// TwinCAT 3 PLC project PLC
// ProgramVersion: 3.1.4024.0
// libraries:
//   SPT Base Types, * (Beckhoff Automation LLC)
//   SPT Event Logger, * (Beckhoff Automation LLC)
//   Tc2_Standard, * (Beckhoff Automation GmbH)
//   Tc2_System, * (Beckhoff Automation GmbH)
//   Tc3_EventLogger, * (Beckhoff Automation GmbH)
//   Tc3_Module, * (Beckhoff Automation GmbH)
//   Tc3_PackML_V2, * (Beckhoff Automation GmbH)
// project tree:
//   / PlcTask.TcTTO (not stored)
//   POUs/ Component.TcPOU, EquipmentModule.TcPOU, EquipmentModuleWithSubModule.TcPOU, Machine.TcPOU, MAIN.TcPOU
// real-time tasks:
//   TASK PlcTask: cycle T#10ms, priority 20, ADS port 350

// ---- POUs/Component.TcPOU
FUNCTION_BLOCK Component EXTENDS FB_ComponentBase
VAR
	ComponentAlarms : ARRAY[1..COMPONENT_ALARM_COUNT] OF FB_TcAlarm;
	testCritical	: BOOL;
	testError		: BOOL;
	testWarning		: BOOL;
	testInfo		: BOOL;
	testVerbose		: BOOL;
	clearAlarms		: BOOL;
	testAnalog		: BOOL;
	AnalogIn		: INT;
END_VAR

VAR CONSTANT
	COMPONENT_ALARM_COUNT : UDINT := 7; //First is InitReferenceEvent
END_VAR

METHOD ChangeEventSeverity
VAR_INPUT
	AlarmID : E_ComponentEvents;
	Severity : TcEventSeverity;
END_VAR
VAR
	localAlarm : TcEventEntry;
END_VAR
localAlarm			 := TC_EVENTS.ComponentEvents.AnalogInAlarm;
localAlarm.eSeverity := Severity;
ComponentAlarms[AlarmID].CreateEx(localAlarm, 0, 0);
END_METHOD

//! @summary Initializes event function blocks using this components's name
METHOD PROTECTED CreateEvents

//! @description This method is called by <c>Initialize()</c> as required
F_CreateAllEventsInClass(Alarms		:= ComponentAlarms,
						 ClassSize	:= SIZEOF(TC_Events.ComponentEvents),
						 pInitEvent := ADR(TC_EVENTS.ComponentEvents.InitReferenceEvent),
						 Prefix		:= Name);

SUPER^.CreateEvents();
END_METHOD

//! @summary This method serves as the entry point for all underlying FB logic
METHOD PUBLIC CyclicLogic

//! @description This method should be called cyclically by descendant function blocks by invoking <c>SUPER^.CyclicLogic()</c>.  Alternatively, the contents of this method could be reimplemented entirely in which case a call to this method would not be necessary.
VAR

END_VAR
IF NOT _InitComplete THEN
	_InitComplete := Initialize();
	RETURN;
END_IF



SUPER^.CyclicLogic();

(*
*
*		Code must be after SUPER^.CyclicLogic();
*
*)

(* Update alarm severity from this component *)
_CurrentAlarmSeverity := F_GetMaxSeverityRaised(Alarms := ComponentAlarms, CurrentSeverity := _CurrentAlarmSeverity);
_Error				  := _CurrentAlarmSeverity >= TcEventSeverity.Error;
END_METHOD

//! @summary Basic component initialization logic
METHOD PROTECTED Initialize : BOOL;

//! @description This method is called by <c>CyclicLogic()</c> as required
Initialize := SUPER^.Initialize();
END_METHOD

//! Provides basic error detection and event handling for this component
METHOD PROTECTED Monitoring

(*! @descriptionThis method is called cyclically by <c>CyclicLogic()</c>*)
VAR

END_VAR
_Busy := FALSE;

//AlarmMonitoring
IF testVerbose AND NOT ComponentAlarms[E_ComponentEvents.VerboseEvent].bRaised THEN
	RaiseAlarm2Args(ComponentAlarms[E_ComponentEvents.VerboseEvent], 'Note 1', 'Note 2');
END_IF

IF testInfo AND NOT ComponentAlarms[E_ComponentEvents.InfoEvent].bRaised THEN
	RaiseAlarm2Args(ComponentAlarms[E_ComponentEvents.InfoEvent], 'Note 1', 'Note 2');
END_IF

IF testWarning AND NOT ComponentAlarms[E_ComponentEvents.WarningEvent].bRaised THEN
	RaiseAlarm2Args(ComponentAlarms[E_ComponentEvents.WarningEvent], 'Note 1', 'Note 2');
END_IF

IF testError AND NOT ComponentAlarms[E_ComponentEvents.ErrorEvent].bRaised THEN
	RaiseAlarm2Args(ComponentAlarms[E_ComponentEvents.ErrorEvent], 'Note 1', 'Note 2');
END_IF

IF testCritical AND NOT ComponentAlarms[E_ComponentEvents.CriticalEvent].bRaised THEN
	RaiseAlarm2Args(ComponentAlarms[E_ComponentEvents.CriticalEvent], 'Note 1', 'Note 2');
END_IF

//Analog Input with Changing Event Severities
IF testAnalog AND NOT ComponentAlarms[E_ComponentEvents.AnalogInAlarm].bRaised THEN
	CASE AnalogIn OF
		0..10:
			ChangeEventSeverity(E_ComponentEvents.AnalogInAlarm, TcEventSeverity.Critical);

		11..100:
			ChangeEventSeverity(E_ComponentEvents.AnalogInAlarm, TcEventSeverity.Error);

		101..999:
			ChangeEventSeverity(E_ComponentEvents.AnalogInAlarm, TcEventSeverity.Info);

		1000..1100:
			ChangeEventSeverity(E_ComponentEvents.AnalogInAlarm, TcEventSeverity.Error);

		1101..1201:
			ChangeEventSeverity(E_ComponentEvents.AnalogInAlarm, TcEventSeverity.Critical);
	END_CASE

	RaiseAlarm2Args(ComponentAlarms[E_ComponentEvents.AnalogInAlarm], 'Analong Input:', TO_STRING(AnalogIn));
ELSIF NOT testAnalog AND_THEN ComponentAlarms[E_ComponentEvents.AnalogInAlarm].bRaised THEN
	ComponentAlarms[E_ComponentEvents.AnalogInAlarm].Clear(0, 0);
END_IF

SUPER^.Monitoring();
END_METHOD

METHOD RaiseAlarm2Args
VAR_IN_OUT
	Alarm : FB_TcAlarm; //Alarm to be raised
END_VAR

VAR_INPUT
	String_1 : STRING; //First String Parameter (The Name of this component will be applied first automatically)
	String_2 : STRING; //Second String Parameter
END_VAR
F_RaiseAlarmWithStringParameters(Alarm	  := Alarm,
								 String_1 := Name,
								 String_2 := String_1,
								 String_3 := String_2);
END_METHOD

//! @summary Clears error flags and error IDs for this component
//Typically called by the EMs SUPER^.Clearing Method
METHOD PUBLIC Reset : BOOL
F_ClearAllEventsInClass(Alarms := ComponentAlarms);
IF SUPER^.Reset() THEN
	_Error	 := FALSE;
	_ErrorID := 0;
	Reset	 := TRUE;
END_IF
END_METHOD

END_FUNCTION_BLOCK

// ---- POUs/EquipmentModule.TcPOU
FUNCTION_BLOCK EquipmentModule EXTENDS FB_PackML_BaseModule
VAR
	//Component
	ComponentOne	: Component := (Name := 'Component One');
	EquipmentAlarms : ARRAY[1..EQUIPMENT_ALARM_COUNT] OF FB_TcAlarm;
	testCritical	: BOOL;
	testError		: BOOL;
	testWarning		: BOOL;
	testInfo		: BOOL;
	testVerbose		: BOOL;
	clearAlarms		: BOOL;

END_VAR

VAR CONSTANT
	EQUIPMENT_ALARM_COUNT : UDINT := 6; //First is InitReferenceEvent
END_VAR

METHOD PROTECTED Clearing
VAR
	i				: UDINT;
	SubModulesReady : BOOL := TRUE;
END_VAR
F_ClearAllEventsInClass(Alarms := EquipmentAlarms);
SUPER^.Clearing();
END_METHOD

//! @summary Initializes event function blocks using this module's name
METHOD PROTECTED CreateEvents

//! @description This method is called by <c>Initialize()</c> as required
F_CreateAllEventsInClass(Alarms		:= EquipmentAlarms,
						 ClassSize	:= SIZEOF(TC_Events.EquipmentModuleEvents),
						 pInitEvent := ADR(TC_EVENTS.EquipmentModuleEvents.InitReferenceEvent),
						 Prefix		:= Name);

SUPER^.CreateEvents();
END_METHOD

//! @summary This method serves as the entry point for all underlying FB logic

//! @description This method should be called cyclically by descendant function blocks by invoking <c>SUPER^.CyclicLogic()</c>.  Alternatively, the contents of this method could be reimplemented entirely in which case a call to this method would not be necessary.
METHOD PUBLIC CyclicLogic
VAR
	i : UDINT;
END_VAR
IF NOT _InitComplete THEN
	_InitComplete := Initialize();
	RETURN;
END_IF

//AlarmHandling();
IF testVerbose AND_THEN NOT EquipmentAlarms[E_EquipmentModuleEvents.VerboseEvent].bRaised THEN
	RaiseAlarm2Args(EquipmentAlarms[E_EquipmentModuleEvents.VerboseEvent], 'Note 1', 'Note 2');
ELSIF NOT testVerbose AND_THEN EquipmentAlarms[E_EquipmentModuleEvents.VerboseEvent].bRaised THEN
	EquipmentAlarms[E_EquipmentModuleEvents.VerboseEvent].Clear(0,0);
END_IF

IF testInfo AND_THEN NOT EquipmentAlarms[E_EquipmentModuleEvents.InfoEvent].bRaised THEN
	RaiseAlarm2Args(EquipmentAlarms[E_EquipmentModuleEvents.InfoEvent], 'Note 1', 'Note 2');
ELSIF NOT testInfo AND_THEN EquipmentAlarms[E_EquipmentModuleEvents.InfoEvent].bRaised THEN
	EquipmentAlarms[E_EquipmentModuleEvents.InfoEvent].Clear(0,0);
END_IF

IF testWarning AND_THEN NOT EquipmentAlarms[E_EquipmentModuleEvents.WarningEvent].bRaised THEN
	RaiseAlarm2Args(EquipmentAlarms[E_EquipmentModuleEvents.WarningEvent], 'Note 1', 'Note 2');
ELSIF NOT testWarning AND_THEN EquipmentAlarms[E_EquipmentModuleEvents.WarningEvent].bRaised THEN
	EquipmentAlarms[E_EquipmentModuleEvents.WarningEvent].Clear(0,0);
END_IF

IF testError AND_THEN NOT EquipmentAlarms[E_EquipmentModuleEvents.ErrorEvent].bRaised THEN
	RaiseAlarm2Args(EquipmentAlarms[E_EquipmentModuleEvents.ErrorEvent], 'Note 1', 'Note 2');
END_IF

IF testCritical AND_THEN NOT EquipmentAlarms[E_EquipmentModuleEvents.CriticalEvent].bRaised THEN
	RaiseAlarm2Args(EquipmentAlarms[E_EquipmentModuleEvents.CriticalEvent], 'Note 1', 'Note 2');
END_IF

SUPER^.CyclicLogic();

(*
*
*		Code must be after SUPER^.CyclicLogic();
*
*)

(* Update alarm severity from this module *)
_CurrentAlarmSeverity := F_GetMaxSeverityRaised(Alarms := EquipmentAlarms, CurrentSeverity := _CurrentAlarmSeverity);
_Error				  := _CurrentAlarmSeverity >= TcEventSeverity.Error;
END_METHOD

//! @summary Basic module initialization logic
METHOD PROTECTED Initialize : BOOL;
VAR
	i						 : UDINT;
	varInfo					 : __SYSTEM.VAR_INFO;
	AllSubUnitsInitialized	 : BOOL := TRUE;
	AllComponentsInitialized : BOOL := TRUE;
END_VAR

//! @description This method is called by <c>CyclicLogic()</c> as required
Initialize := FALSE;
CASE DescendantSequenceState OF
	0:
		LogModeChanges	:= FALSE;
		LogStateChanges := FALSE;

		//Register Submodules

		//Register Components
		RegisterComponent(Component := ComponentOne);
		DescendantSequenceState := DescendantSequenceState + 10;

	10:
		IF SUPER^.Initialize() THEN
			Initialize := TRUE;
		END_IF
END_CASE
END_METHOD

METHOD RaiseAlarm2Args
VAR_IN_OUT
	Alarm : FB_TcAlarm; //Alarm to be raised
END_VAR

VAR_INPUT
	String_1 : STRING; //First String Parameter (The Name of this component will be applied first automatically)
	String_2 : STRING; //Second String Parameter
END_VAR
F_RaiseAlarmWithStringParameters(Alarm	  := Alarm,
								 String_1 := Name,
								 String_2 := String_1,
								 String_3 := String_2);
END_METHOD

END_FUNCTION_BLOCK

// ---- POUs/EquipmentModuleWithSubModule.TcPOU
FUNCTION_BLOCK EquipmentModuleWithSubModule EXTENDS FB_PackML_BaseModule
VAR
	//SubModule
	SubModule : EquipmentModule := (Name := 'SubModule of EM');

	//Component
	ComponentOne	: Component := (Name := 'Component of EM with Sub');
	EquipmentAlarms : ARRAY[1..EQUIPMENT_ALARM_COUNT] OF FB_TcAlarm;
	testCritical	: BOOL;
	testError		: BOOL;
	testWarning		: BOOL;
	testInfo		: BOOL;
	testVerbose		: BOOL;
	clearAlarms		: BOOL;

END_VAR

VAR CONSTANT
	EQUIPMENT_ALARM_COUNT : UDINT := 6; //First is InitReferenceEvent
END_VAR

METHOD PROTECTED Clearing
VAR
	i				: UDINT;
	SubModulesReady : BOOL := TRUE;
END_VAR
F_ClearAllEventsInClass(Alarms := EquipmentAlarms);
SUPER^.Clearing();
END_METHOD

//! @summary Initializes event function blocks using this module's name
METHOD PROTECTED CreateEvents

//! @description This method is called by <c>Initialize()</c> as required
F_CreateAllEventsInClass(Alarms		:= EquipmentAlarms,
						 ClassSize	:= SIZEOF(TC_Events.EquipmentModuleEvents),
						 pInitEvent := ADR(TC_EVENTS.EquipmentModuleEvents.InitReferenceEvent),
						 Prefix		:= Name);

SUPER^.CreateEvents();
END_METHOD

//! @summary This method serves as the entry point for all underlying FB logic

//! @description This method should be called cyclically by descendant function blocks by invoking <c>SUPER^.CyclicLogic()</c>.  Alternatively, the contents of this method could be reimplemented entirely in which case a call to this method would not be necessary.
METHOD PUBLIC CyclicLogic
VAR
	i : UDINT;
END_VAR
IF NOT _InitComplete THEN
	_InitComplete := Initialize();
	RETURN;
END_IF

//AlarmHandling();
IF testVerbose AND NOT EquipmentAlarms[E_EquipmentModuleEvents.VerboseEvent].bRaised THEN
	RaiseAlarm2Args(EquipmentAlarms[E_EquipmentModuleEvents.VerboseEvent], 'Note 1', 'Note 2');
END_IF

IF testInfo AND NOT EquipmentAlarms[E_EquipmentModuleEvents.InfoEvent].bRaised THEN
	RaiseAlarm2Args(EquipmentAlarms[E_EquipmentModuleEvents.InfoEvent], 'Note 1', 'Note 2');
END_IF

IF testWarning AND NOT EquipmentAlarms[E_EquipmentModuleEvents.WarningEvent].bRaised THEN
	RaiseAlarm2Args(EquipmentAlarms[E_EquipmentModuleEvents.WarningEvent], 'Note 1', 'Note 2');
END_IF

IF testError AND NOT EquipmentAlarms[E_EquipmentModuleEvents.ErrorEvent].bRaised THEN
	RaiseAlarm2Args(EquipmentAlarms[E_EquipmentModuleEvents.ErrorEvent], 'Note 1', 'Note 2');
END_IF

IF testCritical AND NOT EquipmentAlarms[E_EquipmentModuleEvents.CriticalEvent].bRaised THEN
	RaiseAlarm2Args(EquipmentAlarms[E_EquipmentModuleEvents.CriticalEvent], 'Note 1', 'Note 2');
END_IF

SUPER^.CyclicLogic();

(*
*
*		Code must be after SUPER^.CyclicLogic();
*
*)

(* Update alarm severity from this module *)
_CurrentAlarmSeverity := F_GetMaxSeverityRaised(Alarms := EquipmentAlarms, CurrentSeverity := _CurrentAlarmSeverity);
_Error				  := _CurrentAlarmSeverity >= TcEventSeverity.Error;
END_METHOD

//! @summary Basic module initialization logic
METHOD PROTECTED Initialize : BOOL;
VAR
	i						 : UDINT;
	varInfo					 : __SYSTEM.VAR_INFO;
	AllSubUnitsInitialized	 : BOOL := TRUE;
	AllComponentsInitialized : BOOL := TRUE;
END_VAR

//! @description This method is called by <c>CyclicLogic()</c> as required
Initialize := FALSE;
CASE DescendantSequenceState OF
	0:
		LogModeChanges	:= FALSE;
		LogStateChanges := FALSE;

		//Register Submodules

		//Register Components
		RegisterSubmodule(SubModule := SubModule);
		RegisterComponent(Component := ComponentOne);
		DescendantSequenceState := DescendantSequenceState + 10;

	10:
		IF SUPER^.Initialize() THEN
			Initialize := TRUE;
		END_IF
END_CASE
END_METHOD

METHOD RaiseAlarm2Args
VAR_IN_OUT
	Alarm : FB_TcAlarm; //Alarm to be raised
END_VAR

VAR_INPUT
	String_1 : STRING; //First String Parameter (The Name of this component will be applied first automatically)
	String_2 : STRING; //Second String Parameter
END_VAR
F_RaiseAlarmWithStringParameters(Alarm	  := Alarm,
								 String_1 := Name,
								 String_2 := String_1,
								 String_3 := String_2);
END_METHOD

END_FUNCTION_BLOCK

// ---- POUs/Machine.TcPOU
FUNCTION_BLOCK Machine EXTENDS FB_PackML_BaseModule
VAR
	EquipOne	: EquipmentModule := (Name := 'Equip One');
	EquipTwo	: EquipmentModuleWithSubModule := (Name := 'Equip Two');
	ComponentMM : Component		  := (Name := 'Component MM');

	//Alarms
	MachineAlarms : ARRAY[1..MACHINE_ALARM_COUNT] OF FB_TcAlarm;
	testCritical  : BOOL;
	testError	  : BOOL;
	testWarning	  : BOOL;
	testInfo	  : BOOL;
	testVerbose	  : BOOL;
	clearAlarms	  : BOOL;
END_VAR

VAR CONSTANT
	MACHINE_ALARM_COUNT : UDINT := 6; //First is InitReferenceEvent
END_VAR

METHOD PROTECTED Clearing
VAR
	i				: UDINT;
	SubModulesReady : BOOL := TRUE;
	ComponentsReady : BOOL := TRUE;
END_VAR
(*
If there are no Components of the Machine
then we can clear the Machine Alarms and let the SUPER handle the rest.

But if the Machine Module has a component
then the process of clearing the alarms 
must be handled in a slightly different manner.
This will prevent an existing alarm condition that is still TRUE
from being cleared and raised multiple times.
*)
IF NumberOfComponents = 0 THEN
	F_ClearAllEventsInClass(Alarms := MachineAlarms);
	SUPER^.Clearing();
ELSE
	CASE SequenceState OF
		0:
			F_ClearAllEventsInClass(Alarms := MachineAlarms);
			SequenceState := SequenceState + 10;

		10:
			FOR i := 1 TO NumberOfSubModules DO
				ipSubModules[i].StateCommand := ePMLCommand_Clear;
			END_FOR

			IF BaseAlarms[E_BaseAlarms.ComponentError].bRaised THEN
				BaseAlarms[E_BaseAlarms.ComponentError].Clear(0, 0);
			END_IF;

			IF BaseAlarms[E_BaseAlarms.SubModuleError].bRaised THEN
				BaseAlarms[E_BaseAlarms.SubModuleError].Clear(0, 0);
			END_IF;

			SequenceState := SequenceState + 10;

		20:
			FOR i := 1 TO NumberOfComponents DO
				IF Parameters_PackML_Base.RESET_COMPONENTS_WITHOUT_ERROR THEN
					ipComponents[i].Reset();
				ELSE
					IF ipComponents[i].Error THEN
						ipComponents[i].Reset();
					END_IF
				END_IF
			END_FOR

			FOR i := 1 TO NumberOfComponents DO
				ComponentsReady := ComponentsReady AND NOT ipComponents[i].Error;
			END_FOR

			IF ComponentsReady THEN
				SequenceState := SequenceState + 10;
			END_IF

		30:
			FOR i := 1 TO NumberOfSubModules DO
				SubModulesReady := SubModulesReady AND (ipSubModules[i].CurrentState = ePMLState_Stopped);
			END_FOR

			IF SubModulesReady AND (StateTasksComplete OR NoStateTasksToComplete) THEN
				NoStateTasksToComplete := TRUE;
				StateTasksComplete	   := FALSE;
				StateComplete();
			END_IF
	END_CASE
END_IF
END_METHOD

//! @summary Initializes event function blocks using this module's name
METHOD PROTECTED CreateEvents

//! @description This method is called by <c>Initialize()</c> as required
F_CreateAllEventsInClass(Alarms		:= MachineAlarms,
						 ClassSize	:= SIZEOF(TC_Events.MachineEvents),
						 pInitEvent := ADR(TC_EVENTS.MachineEvents.InitReferenceEvent),
						 Prefix		:= Name);

SUPER^.CreateEvents();
END_METHOD

//! @summary This method serves as the entry point for all underlying FB logic

//! @description This method should be called cyclically by descendant function blocks by invoking <c>SUPER^.CyclicLogic()</c>.  Alternatively, the contents of this method could be reimplemented entirely in which case a call to this method would not be necessary.
METHOD PUBLIC CyclicLogic
VAR
	i : UDINT;
END_VAR
IF NOT _InitComplete THEN
	_InitComplete := Initialize();
	RETURN;
END_IF

//AlarmHandling();
IF testVerbose AND NOT MachineAlarms[E_MachineEvents.VerboseEvent].bRaised THEN
	RaiseAlarm2Args(MachineAlarms[E_MachineEvents.VerboseEvent], 'Note 1', 'Note 2');
END_IF

IF testCritical AND NOT MachineAlarms[E_MachineEvents.CriticalEvent].bRaised THEN
	RaiseAlarm2Args(MachineAlarms[E_MachineEvents.CriticalEvent], 'Note 1', 'Note 2');
END_IF

//The MachineMonitor is based on the SubModuleMonitor, but is only monitors itself
MachineMonitor();

//
SUPER^.CyclicLogic();

(*
*
*		Code must be after SUPER^.CyclicLogic();
*
*)

(* Update alarm severity from this module *)
_CurrentAlarmSeverity := F_GetMaxSeverityRaised(Alarms := MachineAlarms, CurrentSeverity := _CurrentAlarmSeverity);
_Error				  := _CurrentAlarmSeverity >= TcEventSeverity.Error;


Trace(Message:='Test Mesage');
END_METHOD

//! @summary Basic module initialization logic
METHOD PROTECTED Initialize : BOOL;
VAR
	i						 : UDINT;
	varInfo					 : __SYSTEM.VAR_INFO;
	AllSubUnitsInitialized	 : BOOL := TRUE;
	AllComponentsInitialized : BOOL := TRUE;
END_VAR

//! @description This method is called by <c>CyclicLogic()</c> as required
Initialize := FALSE;
CASE DescendantSequenceState OF
	0:
		LogModeChanges	:= FALSE;
		LogStateChanges := FALSE;

		//Register Submodules
		RegisterSubmodule(EquipOne);
		RegisterSubmodule(EquipTwo);		
		RegisterComponent(ComponentMM);
		DescendantSequenceState := DescendantSequenceState + 10;

	10:
		IF SUPER^.Initialize() THEN
			Initialize := TRUE;
		END_IF
END_CASE
END_METHOD

METHOD MachineMonitor
VAR
	AlarmResponses : ARRAY[0..4] OF E_AlarmResponse; //Temporary response array	
	i			   : UDINT;
END_VAR
IF _CurrentState <> E_PMLState.ePMLState_Aborted AND _CurrentState <> E_PMLState.ePMLState_Aborting AND _CurrentState <> E_PMLState.ePMLState_Clearing AND _CurrentState <> E_PMLState.ePMLState_Stopped AND _CurrentState <> E_PMLState.ePMLState_Stopping THEN
	AlarmResponses := ParentResponseDefinitions;
	CASE AlarmResponses[_CurrentAlarmSeverity] OF
		E_AlarmResponse.Abort_ImmediateError:
			AbortImmediateError(Name, TRUE);

		E_AlarmResponse.Abort_Immediate:
			AbortImmediate();

		E_AlarmResponse.Stop_Immediate:
			StopImmediate();

		E_AlarmResponse.Stop_Controlled:
			StopControlled();

		E_AlarmResponse.Hold_Immediate:
			HoldImmediate();

		E_AlarmResponse.Hold_Controlled:
			HoldControlled();

		E_AlarmResponse.Suspend_Immediate:
			SuspendImmediate();

		E_AlarmResponse.Suspend_Controlled:
			SuspendControlled();

		E_AlarmResponse.NoResponse:
			;
	END_CASE
ELSIF _CurrentState = E_PMLState.ePMLState_Stopped OR _CurrentState = E_PMLState.ePMLState_Stopping THEN
	AlarmResponses := ParentResponseDefinitions;
	CASE AlarmResponses[CurrentAlarmSeverity] OF
		E_AlarmResponse.Abort_ImmediateError:
			AbortImmediateError(Name, TRUE);

		E_AlarmResponse.Abort_Immediate:
			AbortImmediate();

		E_AlarmResponse.NoResponse:
			;
	END_CASE
END_IF
END_METHOD

METHOD RaiseAlarm2Args
VAR_IN_OUT
	Alarm : FB_TcAlarm; //Alarm to be raised
END_VAR

VAR_INPUT
	String_1 : STRING; //First String Parameter (The Name of this component will be applied first automatically)
	String_2 : STRING; //Second String Parameter
END_VAR
F_RaiseAlarmWithStringParameters(Alarm	  := Alarm,
								 String_1 := Name,
								 String_2 := String_1,
								 String_3 := String_2);
END_METHOD

END_FUNCTION_BLOCK

// ---- POUs/MAIN.TcPOU
PROGRAM MAIN
VAR
	Machine			  : Machine := (Name := 'Machine');
	resetStateMachine : BOOL;
	abort			  : BOOL;
	stop			  : BOOL;
END_VAR

// All sample code provided by Beckhoff Automation LLC are for illustrative purposes only and are provided “as is” and without any warranties, express or implied. Actual implementations in applications will vary significantly. Beckhoff Automation LLC shall have no liability for, and does not waive any rights in relation to, any code samples that it provides or the use of such code samples for any purpose.

(*
This sample demonstrates a way to implement alarms for modules and components.
As an incorrect implementation can lead to an endless loop of Raise/CLear it is important to understand when to clear alarms.
Once of the most important details is that the _CurrentAlarmSeverity for a Component/Module must be set locally after the call to SUPER^.CyclicLogic.
This is due to the fact that _CurrentAlarmSeverity is reset to Verbose in the base class.
 

Component
	The Component includes a Monitoring method which is called by the Cyclic Logic of the base class.
	This method includes a test variable for each of the Severity levels (Verbose, Info, Warning, Error, Critical) 
	The default severities are set in the Base Class.

	Additionally, an example for changing the severity at run time is given which changes the based on the value of an pressumed Analog Input.

	Each of these Component Alarms are only cleared when the Module containing the component calls its SUPER^.Clearing()
 
Equipment Module
	The EM CyclicLogic method has code to monitor possible alarm conditions. 
	The EM does not have a Monitoring method in the base class, you can add your own and call it from CyclicLogic.
	Take note that the first 3 alarms (Verbose, Info, Warning) reset themselves once the condition is FALSE, 
	while the Error and Critical alarms are required to be reset from SUPER^.Clearing.

Machine Module
	 Most of the implementation for Alarms in the Machine module are the same as the Equipment Module.
	 The 2 differences are the implementation of a MachineMonitor, which provides similar functionality to the SubModuleMonitor method, 
	 and the way in which the Clearing method is implemented.
	 
	The MachineMonitor method is called by CyclicLogic and is a simplified version of the SubModuleMonitor in the base class,
	the SubModuleMonitor requires a FOR loop to process all of the SubModule, and this is removed from the MachineMonitor.
	
	The Clearing method is based on the one from the base class, but with the addition of a check for any Components of the Machine Module.
	More information is provided in the code.

*)

//This is for debug only and should be removed
_AppInfo.KeepOutputsOnBP := TRUE;

//
Machine.CyclicLogic();

//
CASE Machine.CurrentState OF
	E_PMLState.ePMLState_Aborted:
		IF resetStateMachine THEN
			resetStateMachine := FALSE;
			Machine.ChangeState(State := E_PMLCommand.ePMLCommand_Clear);
		END_IF

	E_PMLState.ePMLState_Stopped:
		Machine.ChangeState(State := E_PMLCommand.ePMLCommand_Reset);

	E_PMLState.ePMLState_Idle:
		Machine.ChangeState(State := E_PMLCommand.ePMLCommand_Start);
END_CASE

//
IF abort THEN
	abort := FALSE;
	Machine.ChangeState(State := E_PMLCommand.ePMLCommand_Abort);
END_IF

IF stop THEN
	stop := FALSE;
	Machine.ChangeState(State := ePMLCommand_Stop);
END_IF

END_PROGRAM
